{region '#Template'}
	{attribute 'Version' := '5.1.0.0'}
	{attribute 'Tags' := '"LCID": "1031", "Text": "AC, Allgemein, AHU, Betriebsart"'}
	{attribute 'Tags' := '"LCID": "1033", "Text": "AC, General, AHU, Operating mode"'}
	{attribute 'Using' := '"Type": "Template", "URI": "E_BA_AC_OpMod01"'}
	{attribute 'Description' := '"LCID": "1031", "Text": "Betriebsart"'}
	{attribute 'Description' := '"LCID": "1033", "Text": "Operating mode"'}
{endregion}

FUNCTION_BLOCK FB_BA_AC_OpModAggMdlt
VAR_INPUT
	stPriorityEn				: ST_BA_PriorityEn;	
	eOpMode					: E_BA_AC_OpMod01;
	bFdb					: BOOL;
	fDlyOn					: REAL;	
	fDlyOff					: REAL;	
END_VAR
VAR_OUTPUT
	stCmd					: ST_BA_Mdlt;
	nRemSecStepUp           : UDINT;
	nRemSecStepDown         : UDINT;
END_VAR
VAR_IN_OUT
	stStep					: ST_BA_Step;
END_VAR
VAR_INPUT CONSTANT
	OpModVal				: FB_BA_MMUX_UDI16;
	DelayOn					: FB_BA_MMUX_B16;
	DelayOff				: FB_BA_MMUX_B16;
	IgnoreFdb				: FB_BA_MMUX_B16;	
	Step                    : FB_BA_StepMdlt;
END_VAR
VAR_INPUT CONSTANT PERSISTENT
	bInit					: BOOL := TRUE;
	arrOpModVal				: ARRAY [1..16] OF E_BA_Mdlt;
	arrIgnoreDelayOnVal 	: ARRAY [1..16] OF BOOL;
	arrIgnoreDelayOffVal	: ARRAY [1..16] OF BOOL;
	arrIgnoreFdbVal 		: ARRAY [1..16] OF BOOL;	
END_VAR
VAR
	eVal					: E_BA_Mdlt;
	_bFdb					: BOOL;	
	nDelayOn				: UDINT;
	nDelayOff				: UDINT;	
END_VAR
VAR // added by the converter: edge detectors and wires of the graphical bodies
    _w1, _w2 : UDINT;
END_VAR

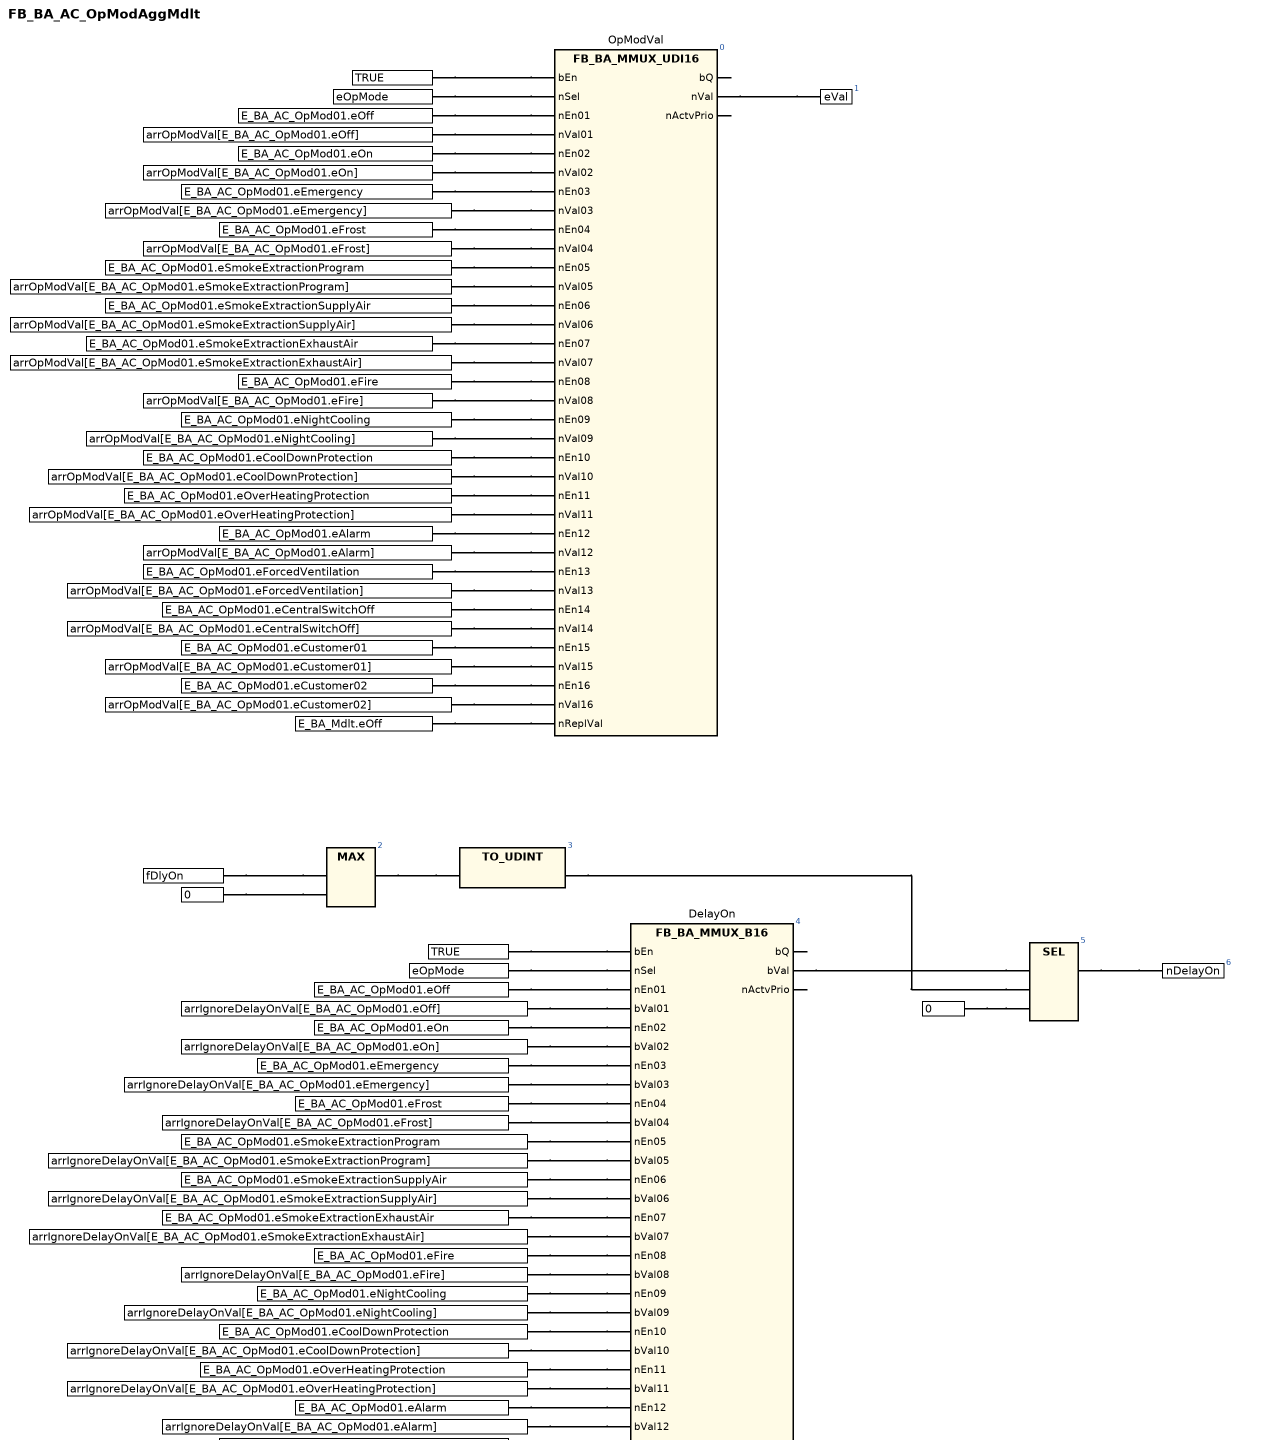
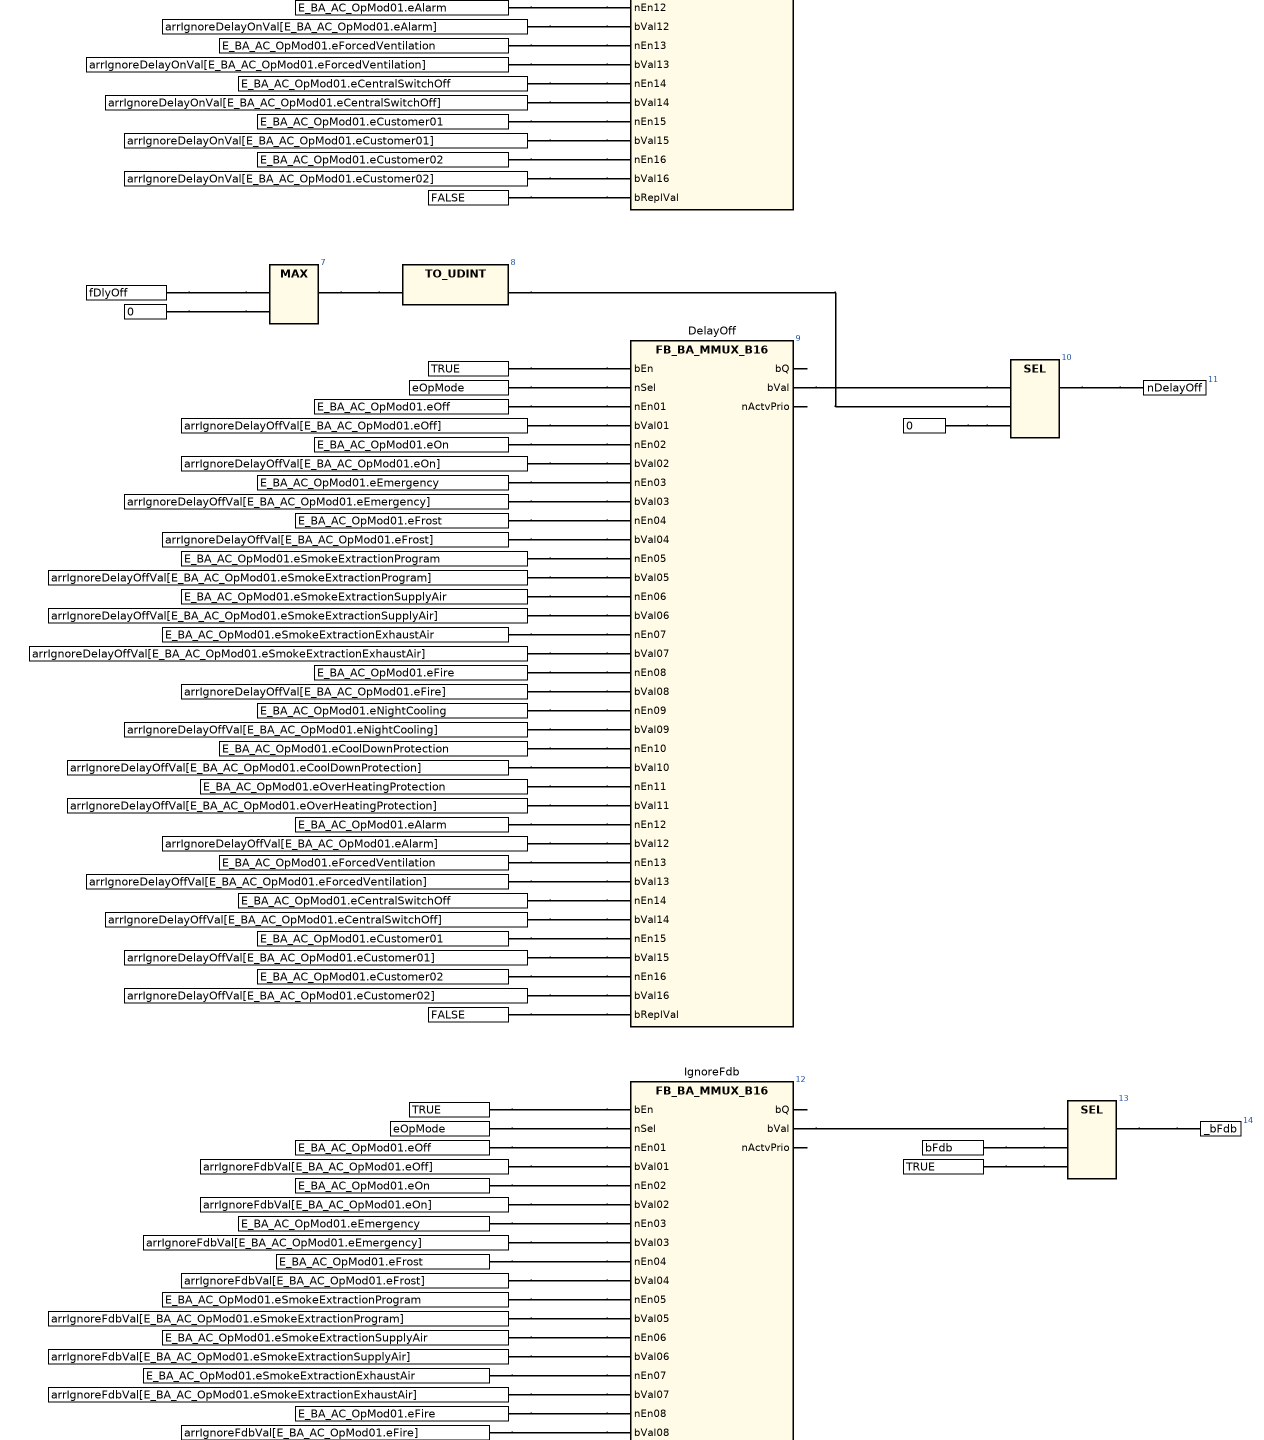
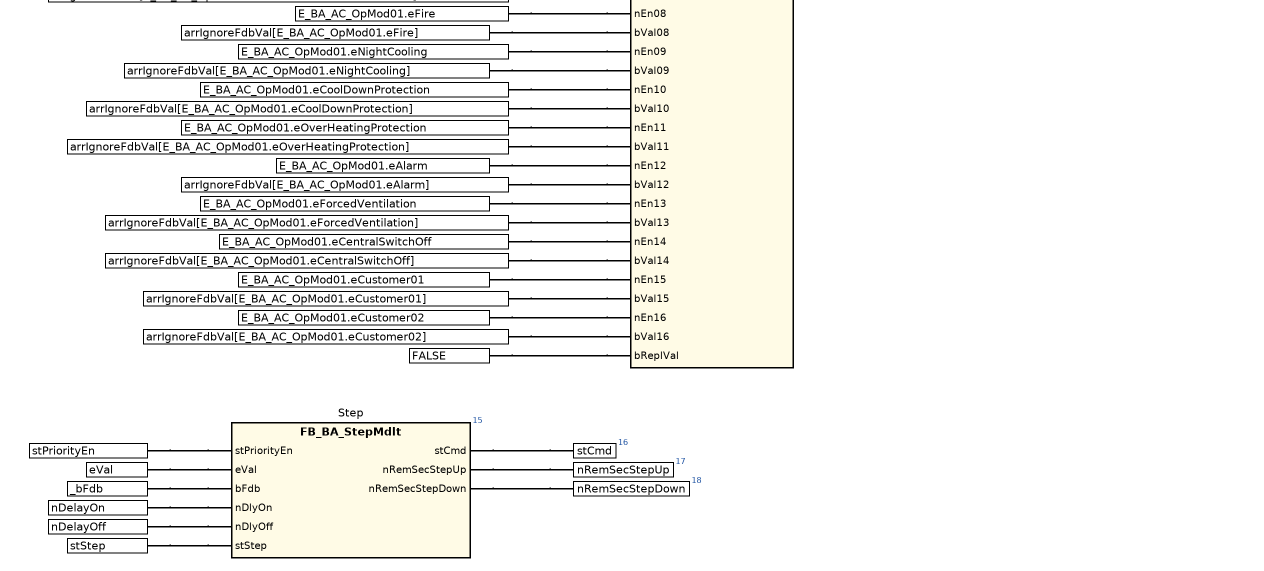
OpModVal(
    bEn := TRUE,
    nSel := eOpMode,
    nEn01 := E_BA_AC_OpMod01.eOff,
    nVal01 := arrOpModVal[E_BA_AC_OpMod01.eOff],
    nEn02 := E_BA_AC_OpMod01.eOn,
    nVal02 := arrOpModVal[E_BA_AC_OpMod01.eOn],
    nEn03 := E_BA_AC_OpMod01.eEmergency,
    nVal03 := arrOpModVal[E_BA_AC_OpMod01.eEmergency],
    nEn04 := E_BA_AC_OpMod01.eFrost,
    nVal04 := arrOpModVal[E_BA_AC_OpMod01.eFrost],
    nEn05 := E_BA_AC_OpMod01.eSmokeExtractionProgram,
    nVal05 := arrOpModVal[E_BA_AC_OpMod01.eSmokeExtractionProgram],
    nEn06 := E_BA_AC_OpMod01.eSmokeExtractionSupplyAir,
    nVal06 := arrOpModVal[E_BA_AC_OpMod01.eSmokeExtractionSupplyAir],
    nEn07 := E_BA_AC_OpMod01.eSmokeExtractionExhaustAir,
    nVal07 := arrOpModVal[E_BA_AC_OpMod01.eSmokeExtractionExhaustAir],
    nEn08 := E_BA_AC_OpMod01.eFire,
    nVal08 := arrOpModVal[E_BA_AC_OpMod01.eFire],
    nEn09 := E_BA_AC_OpMod01.eNightCooling,
    nVal09 := arrOpModVal[E_BA_AC_OpMod01.eNightCooling],
    nEn10 := E_BA_AC_OpMod01.eCoolDownProtection,
    nVal10 := arrOpModVal[E_BA_AC_OpMod01.eCoolDownProtection],
    nEn11 := E_BA_AC_OpMod01.eOverHeatingProtection,
    nVal11 := arrOpModVal[E_BA_AC_OpMod01.eOverHeatingProtection],
    nEn12 := E_BA_AC_OpMod01.eAlarm,
    nVal12 := arrOpModVal[E_BA_AC_OpMod01.eAlarm],
    nEn13 := E_BA_AC_OpMod01.eForcedVentilation,
    nVal13 := arrOpModVal[E_BA_AC_OpMod01.eForcedVentilation],
    nEn14 := E_BA_AC_OpMod01.eCentralSwitchOff,
    nVal14 := arrOpModVal[E_BA_AC_OpMod01.eCentralSwitchOff],
    nEn15 := E_BA_AC_OpMod01.eCustomer01,
    nVal15 := arrOpModVal[E_BA_AC_OpMod01.eCustomer01],
    nEn16 := E_BA_AC_OpMod01.eCustomer02,
    nVal16 := arrOpModVal[E_BA_AC_OpMod01.eCustomer02],
    nReplVal := E_BA_Mdlt.eOff); // FB_BA_MMUX_UDI16
eVal := OpModVal.nVal;
_w1 := TO_UDINT(MAX(fDlyOn, 0));
DelayOn(
    bEn := TRUE,
    nSel := eOpMode,
    nEn01 := E_BA_AC_OpMod01.eOff,
    bVal01 := arrIgnoreDelayOnVal[E_BA_AC_OpMod01.eOff],
    nEn02 := E_BA_AC_OpMod01.eOn,
    bVal02 := arrIgnoreDelayOnVal[E_BA_AC_OpMod01.eOn],
    nEn03 := E_BA_AC_OpMod01.eEmergency,
    bVal03 := arrIgnoreDelayOnVal[E_BA_AC_OpMod01.eEmergency],
    nEn04 := E_BA_AC_OpMod01.eFrost,
    bVal04 := arrIgnoreDelayOnVal[E_BA_AC_OpMod01.eFrost],
    nEn05 := E_BA_AC_OpMod01.eSmokeExtractionProgram,
    bVal05 := arrIgnoreDelayOnVal[E_BA_AC_OpMod01.eSmokeExtractionProgram],
    nEn06 := E_BA_AC_OpMod01.eSmokeExtractionSupplyAir,
    bVal06 := arrIgnoreDelayOnVal[E_BA_AC_OpMod01.eSmokeExtractionSupplyAir],
    nEn07 := E_BA_AC_OpMod01.eSmokeExtractionExhaustAir,
    bVal07 := arrIgnoreDelayOnVal[E_BA_AC_OpMod01.eSmokeExtractionExhaustAir],
    nEn08 := E_BA_AC_OpMod01.eFire,
    bVal08 := arrIgnoreDelayOnVal[E_BA_AC_OpMod01.eFire],
    nEn09 := E_BA_AC_OpMod01.eNightCooling,
    bVal09 := arrIgnoreDelayOnVal[E_BA_AC_OpMod01.eNightCooling],
    nEn10 := E_BA_AC_OpMod01.eCoolDownProtection,
    bVal10 := arrIgnoreDelayOnVal[E_BA_AC_OpMod01.eCoolDownProtection],
    nEn11 := E_BA_AC_OpMod01.eOverHeatingProtection,
    bVal11 := arrIgnoreDelayOnVal[E_BA_AC_OpMod01.eOverHeatingProtection],
    nEn12 := E_BA_AC_OpMod01.eAlarm,
    bVal12 := arrIgnoreDelayOnVal[E_BA_AC_OpMod01.eAlarm],
    nEn13 := E_BA_AC_OpMod01.eForcedVentilation,
    bVal13 := arrIgnoreDelayOnVal[E_BA_AC_OpMod01.eForcedVentilation],
    nEn14 := E_BA_AC_OpMod01.eCentralSwitchOff,
    bVal14 := arrIgnoreDelayOnVal[E_BA_AC_OpMod01.eCentralSwitchOff],
    nEn15 := E_BA_AC_OpMod01.eCustomer01,
    bVal15 := arrIgnoreDelayOnVal[E_BA_AC_OpMod01.eCustomer01],
    nEn16 := E_BA_AC_OpMod01.eCustomer02,
    bVal16 := arrIgnoreDelayOnVal[E_BA_AC_OpMod01.eCustomer02],
    bReplVal := FALSE); // FB_BA_MMUX_B16
nDelayOn := SEL(DelayOn.bVal, _w1, 0);
_w2 := TO_UDINT(MAX(fDlyOff, 0));
DelayOff(
    bEn := TRUE,
    nSel := eOpMode,
    nEn01 := E_BA_AC_OpMod01.eOff,
    bVal01 := arrIgnoreDelayOffVal[E_BA_AC_OpMod01.eOff],
    nEn02 := E_BA_AC_OpMod01.eOn,
    bVal02 := arrIgnoreDelayOffVal[E_BA_AC_OpMod01.eOn],
    nEn03 := E_BA_AC_OpMod01.eEmergency,
    bVal03 := arrIgnoreDelayOffVal[E_BA_AC_OpMod01.eEmergency],
    nEn04 := E_BA_AC_OpMod01.eFrost,
    bVal04 := arrIgnoreDelayOffVal[E_BA_AC_OpMod01.eFrost],
    nEn05 := E_BA_AC_OpMod01.eSmokeExtractionProgram,
    bVal05 := arrIgnoreDelayOffVal[E_BA_AC_OpMod01.eSmokeExtractionProgram],
    nEn06 := E_BA_AC_OpMod01.eSmokeExtractionSupplyAir,
    bVal06 := arrIgnoreDelayOffVal[E_BA_AC_OpMod01.eSmokeExtractionSupplyAir],
    nEn07 := E_BA_AC_OpMod01.eSmokeExtractionExhaustAir,
    bVal07 := arrIgnoreDelayOffVal[E_BA_AC_OpMod01.eSmokeExtractionExhaustAir],
    nEn08 := E_BA_AC_OpMod01.eFire,
    bVal08 := arrIgnoreDelayOffVal[E_BA_AC_OpMod01.eFire],
    nEn09 := E_BA_AC_OpMod01.eNightCooling,
    bVal09 := arrIgnoreDelayOffVal[E_BA_AC_OpMod01.eNightCooling],
    nEn10 := E_BA_AC_OpMod01.eCoolDownProtection,
    bVal10 := arrIgnoreDelayOffVal[E_BA_AC_OpMod01.eCoolDownProtection],
    nEn11 := E_BA_AC_OpMod01.eOverHeatingProtection,
    bVal11 := arrIgnoreDelayOffVal[E_BA_AC_OpMod01.eOverHeatingProtection],
    nEn12 := E_BA_AC_OpMod01.eAlarm,
    bVal12 := arrIgnoreDelayOffVal[E_BA_AC_OpMod01.eAlarm],
    nEn13 := E_BA_AC_OpMod01.eForcedVentilation,
    bVal13 := arrIgnoreDelayOffVal[E_BA_AC_OpMod01.eForcedVentilation],
    nEn14 := E_BA_AC_OpMod01.eCentralSwitchOff,
    bVal14 := arrIgnoreDelayOffVal[E_BA_AC_OpMod01.eCentralSwitchOff],
    nEn15 := E_BA_AC_OpMod01.eCustomer01,
    bVal15 := arrIgnoreDelayOffVal[E_BA_AC_OpMod01.eCustomer01],
    nEn16 := E_BA_AC_OpMod01.eCustomer02,
    bVal16 := arrIgnoreDelayOffVal[E_BA_AC_OpMod01.eCustomer02],
    bReplVal := FALSE); // FB_BA_MMUX_B16
nDelayOff := SEL(DelayOff.bVal, _w2, 0);
IgnoreFdb(
    bEn := TRUE,
    nSel := eOpMode,
    nEn01 := E_BA_AC_OpMod01.eOff,
    bVal01 := arrIgnoreFdbVal[E_BA_AC_OpMod01.eOff],
    nEn02 := E_BA_AC_OpMod01.eOn,
    bVal02 := arrIgnoreFdbVal[E_BA_AC_OpMod01.eOn],
    nEn03 := E_BA_AC_OpMod01.eEmergency,
    bVal03 := arrIgnoreFdbVal[E_BA_AC_OpMod01.eEmergency],
    nEn04 := E_BA_AC_OpMod01.eFrost,
    bVal04 := arrIgnoreFdbVal[E_BA_AC_OpMod01.eFrost],
    nEn05 := E_BA_AC_OpMod01.eSmokeExtractionProgram,
    bVal05 := arrIgnoreFdbVal[E_BA_AC_OpMod01.eSmokeExtractionProgram],
    nEn06 := E_BA_AC_OpMod01.eSmokeExtractionSupplyAir,
    bVal06 := arrIgnoreFdbVal[E_BA_AC_OpMod01.eSmokeExtractionSupplyAir],
    nEn07 := E_BA_AC_OpMod01.eSmokeExtractionExhaustAir,
    bVal07 := arrIgnoreFdbVal[E_BA_AC_OpMod01.eSmokeExtractionExhaustAir],
    nEn08 := E_BA_AC_OpMod01.eFire,
    bVal08 := arrIgnoreFdbVal[E_BA_AC_OpMod01.eFire],
    nEn09 := E_BA_AC_OpMod01.eNightCooling,
    bVal09 := arrIgnoreFdbVal[E_BA_AC_OpMod01.eNightCooling],
    nEn10 := E_BA_AC_OpMod01.eCoolDownProtection,
    bVal10 := arrIgnoreFdbVal[E_BA_AC_OpMod01.eCoolDownProtection],
    nEn11 := E_BA_AC_OpMod01.eOverHeatingProtection,
    bVal11 := arrIgnoreFdbVal[E_BA_AC_OpMod01.eOverHeatingProtection],
    nEn12 := E_BA_AC_OpMod01.eAlarm,
    bVal12 := arrIgnoreFdbVal[E_BA_AC_OpMod01.eAlarm],
    nEn13 := E_BA_AC_OpMod01.eForcedVentilation,
    bVal13 := arrIgnoreFdbVal[E_BA_AC_OpMod01.eForcedVentilation],
    nEn14 := E_BA_AC_OpMod01.eCentralSwitchOff,
    bVal14 := arrIgnoreFdbVal[E_BA_AC_OpMod01.eCentralSwitchOff],
    nEn15 := E_BA_AC_OpMod01.eCustomer01,
    bVal15 := arrIgnoreFdbVal[E_BA_AC_OpMod01.eCustomer01],
    nEn16 := E_BA_AC_OpMod01.eCustomer02,
    bVal16 := arrIgnoreFdbVal[E_BA_AC_OpMod01.eCustomer02],
    bReplVal := FALSE); // FB_BA_MMUX_B16
_bFdb := SEL(IgnoreFdb.bVal, bFdb, TRUE);
Step(
    stPriorityEn := stPriorityEn,
    eVal := eVal,
    bFdb := _bFdb,
    nDlyOn := nDelayOn,
    nDlyOff := nDelayOff,
    stStep := stStep); // FB_BA_StepMdlt
stCmd := Step.stCmd;
nRemSecStepUp := Step.nRemSecStepUp;
nRemSecStepDown := Step.nRemSecStepDown;

END_FUNCTION_BLOCK

(* stored: Version 1.1.0.1, ProductVersion 3.1.4024.12
   POU FB_BA_AC_OpModAggMdlt: Id {d514b2ee-0a7c-45e3-ac57-6bdc77b8ed1d}, SpecialFunc None *)
